Staubli VAL3: tCommande.pgx

program tCommande()
begin
  // Trame attendue depuis le PC :
  // {index;type;x;y;z;rx;ry;rz;vel}
  // type : 0=movej, 1=movel
  // vel  : vitesse TCP mm/s

  while true
    // Attente que la file ne soit pas pleine
    wait(nQueueCount < nQueueSize)

    // Recherche debut de trame
    do
      nNbChar = sioGet(sioSocket, nData)
    until nNbChar > 0 and nData == nSof

    // Lecture des 9 champs
    call getNum(nCmdIndex,                       nDivider)
    call getNum(nCmdType,                        nDivider)
    call getNum(pCmdQueue[nQueueWrite].trsf.x,   nDivider)
    call getNum(pCmdQueue[nQueueWrite].trsf.y,   nDivider)
    call getNum(pCmdQueue[nQueueWrite].trsf.z,   nDivider)
    call getNum(pCmdQueue[nQueueWrite].trsf.rx,  nDivider)
    call getNum(pCmdQueue[nQueueWrite].trsf.ry,  nDivider)
    call getNum(pCmdQueue[nQueueWrite].trsf.rz,  nDivider)
    call getNum(nCmdVel,                         nEof)

    // Ecriture dans la file
    nTypeQueue[nQueueWrite]  = nCmdType
    nIndexQueue[nQueueWrite] = nCmdIndex
    nVelQueue[nQueueWrite]   = nCmdVel

    // Avance le pointeur d ecriture (circulaire)
    nQueueWrite = nQueueWrite + 1
    if nQueueWrite >= nQueueSize
      nQueueWrite = 0
    endIf
    nQueueCount = nQueueCount + 1

    delay(0)
  endWhile
end
